PROGRAM MAIN
VAR
	nCounter : DINT;
END_VAR

nCounter := nCounter +1;

END_PROGRAM

(* stored: Version 1.1.0.1, ProductVersion 3.1.4024.2
   POU MAIN: Id {7ceb935c-a53a-421b-89e2-f98929365a15}, SpecialFunc None *)
